{attribute 'TcGenerated'}
{attribute 'no-analysis'}
{attribute 'linkalways'}
// This function has been automatically generated from the project information.
VAR_GLOBAL CONSTANT
	{attribute 'const_non_replaced'}
	stLibVersion_FM_Common_Interfaces : ST_LibVersion := (iMajor := 0, iMinor := 0, iBuild := 1, iRevision := 0, nFlags := 0, sVersion := '0.0.1');
END_VAR

(* stored: Version 1.1.0.1
   GVL Global_Version: Id {462b9121-315f-0480-3afd-e9196d8f757b} *)
